(* PLC project Generated.project, CODESYS CODESYS V3.5 SP19 Patch 1 *)
(* stored: creationDateTime 2026-08-18T15:58:35.301546, modificationDateTime 2026-08-18T15:58:35.301546 *)

TYPE ST_ChainBucket : STRUCT
  Idx101_BucketIsOpen : BOOL;  (* 1 = Benne Mécaniquement Ouvert | 0 = Non Confirmé *)
  Idx102_BucketIsClosed : BOOL;  (* 1 = Benne Mécaniquement Fermé | 0 = Non Confirmé *)
  Idx103_OffsetPos_M : REAL;  (* [mètres] Écart d'Ouverture Câble M1/M2 *)
  Idx104_AutoSeqActive : BOOL;  (* : 1 = Séquencement auto (ouverture/fermeture armée par mouvement couplé) en cours *)
  Idx105_StateIncoherent : BOOL;  (* : 1 = État ouvert/fermé INCONNU (ni IsOpen ni IsClosed fiable) -- cause fréquente de blocage *)
  Idx106_FBState : E_State;  (* : État machine FB_Bucket (READY/BUSY/DONE/DISABLED) *)
  Idx107_LastPosM2Open_M : REAL;  (* : Dernière position M2 mémorisée "ouvert" *)
  Idx108_LastPosM2Close_M : REAL;  (* : Dernière position M2 mémorisée "fermé" *)
  Idx109_BucketTooOpen : BOOL;  (* ⚠️ Dépassement ouverture : Delta < OffsetOpen - Tolerance (Enrouler M2) *)
  Idx110_BucketTooClosed : BOOL;  (* ⚠️ Dépassement fermeture : Delta > OffsetClose + Tolerance (Dérouler M2) *)
  Idx111_BucketIsIntermediate : BOOL;  (* ↔️ Position intermédiaire (entrebâillée entre ouvert et fermé) *)
  Idx112_DeltaPosition_M : REAL;  (* 📏 Écart réel signé M2 - M1 (mètres) en direct *)
  Idx201_HmiCmd_BtnOpen : BOOL;  (* 1 = Demande Ouverture IHM | 0 = Relâché *)
  Idx202_HmiCmd_BtnClose : BOOL;  (* 1 = Demande Fermeture IHM | 0 = Relâché *)
  Idx203_CycleCmd_Open : BOOL;  (* 1 = Demande Ouverture par le Cycle Auto *)
  Idx204_CoupledDiveOpenArmed : BOOL;  (* : 1 = Ouverture auto armée (descente couplée demandée, benne pas ouverte) *)
  Idx205_CoupledAscentCloseArmed : BOOL;  (* : 1 = Fermeture auto armée (montée couplée demandée, benne pas fermée) *)
  Idx206_CloseReqActive : BOOL;  (* : 1 = Fermeture mémorisée/en cours (instBucket.CloseReq -- reste à 1 si recul partiel non terminé) *)
  Idx207_OpenReqActive : BOOL;  (* : 1 = Ouverture mémorisée/en cours (instBucket.OpenReq -- idem) *)
  Idx208_MotionBlockedByBucket : BOOL;  (* : 1 = Mouvement couplé BLOQUÉ (auto-séquencement armé mais benne pas Busy -- vérifier Idx306_ErrorIdRaw) *)
  Idx301_EmergencyChainClosed : BOOL;  (* 1 = Boucle Urgence OK | 0 = AU Appuyé *)
  Idx302_BucketFaultActive : BOOL;  (* 0 = Sain | 1 = Défaut Mouvement Benne *)
  Idx303_KoboldAutoStopEnabled : BOOL;  (* 1 = Toggle IHM arrêt auto descente actif *)
  Idx304_KoboldImmersionConfirmed : BOOL;  (* : 1 = Immersion confirmée (front Kobold dans la fenêtre) *)
  Idx305_KoboldBottomTouchLatched : BOOL;  (* : 1 = Fond détecté, descente bloquée (ProcessPermitM1/M2_Descend) *)
  Idx306_ErrorIdRaw : WORD;  (* : bitfield brut FB_Bucket (bit0 timeout, bit1 incohérence, bit2 limites, bit3 codeur non référencé, bit4 glissement M1) *)
  Idx401_BucketBusy : BOOL;  (* 1 = Mouvement Mâchoires en cours | 0 = Repos *)
  Idx402_BucketDone : BOOL;  (* 1 = Position Cible Atteinte | 0 = En cours *)
  Idx403_ControlAscentActive : BOOL;  (* : 1 = Phase vitesse contrôlée montée en cours (post-fermeture auto) *)
  Idx501_M2_CmdRev_DQ : BOOL;  (* 1 = Relais Action Benne M2 ON *)
END_STRUCT;
END_TYPE

TYPE ST_ChainContextGlobal : STRUCT
  Idx101_ModeActive : E_Mode;  (* Mode de marche actif (MANUEL, SEMI_AUTO, MAINT_N1, MAINT_N2) *)
  Idx102_SimulationEnabled : BOOL;  (* 0 = Matériel Réel (Nominal) | 1 = SIMULATION ACTIVE ⚠️ *)
  Idx103_JoystickCommOk : BOOL;  (* 1 = Comm CANopen Joystick OK (Sain) | 0 = Perte Comm CAN *)
  Idx201_JoystickSelected : BOOL;  (* 1 = Pilotage par Joystick Hall | 0 = Pilotage par Boutons IHM *)
  Idx202_BypassNetworkGlobal : BOOL;  (* 0 = Comm Réseau OK | 1 = BYPASS RÉSEAU ACTIF ⚠️ *)
  Idx203_BypassSensorsGlobal : BOOL;  (* 0 = Capteurs Actifs | 1 = AU MOINS 1 CAPTEUR SHUNTÉ ⚠️ *)
  Idx301_EmergencyChainClosed : BOOL;  (* 1 = Boucle AU Matérielle Fermée (OK) | 0 = AU APPUYÉ *)
  Idx302_PowerContactorEngaged : BOOL;  (* 1 = Puissance Armée | 0 = Puissance Coupée *)
  Idx303_SafeStopActiveAny : BOOL;  (* 0 = Sain | 1 = AU MOINS UN SAFESTOP MÉTIER ACTIF *)
  Idx304_PowerCutOffActiveAny : BOOL;  (* 0 = Sain | 1 = COUPURE GENERAL COLLAGE ACTIVEE *)
  Idx401_HmiHeartbeatOk : BOOL;  (* 1 = Liaison IHM Active | 0 = Perte Liaison IHM *)
  Idx402_CycleAutoBusy : BOOL;  (* 1 = Séquenceur Auto en Cours | 0 = Repos *)
END_STRUCT;
END_TYPE

(* ======================================================================= 🔄 ST_ChainCycleSemiAuto — Diagnostic chronologique Séquenceur Semi-Auto ─────────────────────────────────────────────────────────────── 🎯 Rôle : Vue dépannage / Watch CODESYS pour le cycle semi-automatique 📄 Doc métier : DOC/AF/AF_Partie-14_Fonction_Troubleshooting/FB_TroubleshootingView_v1.2.md 🔒 Sécurité : 100% lecture seule / diagnostic d'observation ======================================================================= *)
TYPE ST_ChainCycleSemiAuto : STRUCT
  Idx101_ModeSemiAutoActive : BOOL;  (* 🚦 1. Conditions d'engagement et autorisations 1 = Mode arbitré SEMI_AUTO actif | 0 = Autre mode *)
  Idx102_PowerAndSafetyOk : BOOL;  (* 1 = Chaîne de sécurité OK (PowerContactorEngaged) *)
  Idx103_HeartbeatIhmOk : BOOL;  (* 1 = Liaison IHM<->PLC valide *)
  Idx104_DeadmanArmed : BOOL;  (* 1 = Bouton homme-mort armé (fenêtre 3s active) *)
  Idx105_MancheDeflechi : BOOL;  (* 1 = Permis mouvement armé (manche hors zone neutre) *)
  Idx106_HomedM1M2 : BOOL;  (* 1 = Codeurs treuils M1 et M2 référencés *)
  Idx107_StartCycleRequest : BOOL;  (* 1 = Demande Start reçue (IHM) *)
  Idx108_AbortCycleRequest : BOOL;  (* 1 = Demande Abort reçue (IHM) *)
  Idx201_Ready : BOOL;  (* 🔄 2. État du Séquenceur 1 = Séquenceur prêt à démarrer *)
  Idx202_Busy : BOOL;  (* 1 = Cycle en cours d'exécution *)
  Idx203_Done : BOOL;  (* 1 = Cycle terminé avec succès *)
  Idx204_Error : BOOL;  (* 1 = Défaut ou anomalie bloquante sur le cycle *)
  Idx205_ErrorId : WORD;  (* Code d'erreur interne FB_Cycle *)
  Idx206_Step : E_CycleStep;  (* Étape courante (X0 à X13 + STABILIZING) *)
  Idx207_StepStr : STRING(40);  (* Libellé explicite de l'étape *)
  Idx208_StepAtError : E_CycleStep;  (* Étape mémorisée lors du dernier défaut *)
  Idx301_TargetPosition : INT;  (* 🎯 3. Consignes & Feedbacks Opérationnels Cible translation sélectionnée (1=Trémie, 3=P1) *)
  Idx302_TargetDepth_M : REAL;  (* Profondeur de consigne (m) *)
  Idx303_KoboldBottomTouch : BOOL;  (* 1 = Détection contact fond Kobold *)
  Idx304_SpeedMismatchActive : BOOL;  (* 1 = Alerte écart de vitesse M1/M2 active *)
  Idx305_LimitLegalReached : BOOL;  (* 1 = Limite légale atteinte (descente bloquée) *)
  Idx306_WinchSyncError : BOOL;  (* 1 = Erreur de synchronisme M1/M2 *)
END_STRUCT;
END_TYPE

TYPE ST_ChainDredgingAssist : STRUCT
  Idx101_EnableDiveSearch : BOOL;  (* 1 = Assistance Plongée Armée (IHM) | 0 = Désarmée *)
  Idx102_EnableExtractionSequence : BOOL;  (* 1 = Assistance Extraction Armée (IHM) | 0 = Désarmée *)
  Idx103_EnableDumpAtTremie : BOOL;  (* 1 = Mode Vidage Trémie Armé (IHM) | 0 = Désarmé *)
  Idx201_DiveReady : BOOL;  (* 1 = Assistance Plongée Prête | 0 = Non Prête *)
  Idx202_DiveBusy : BOOL;  (* 1 = Séquence Plongée En Cours | 0 = Repos *)
  Idx203_DiveDone : BOOL;  (* 1 = Fond Confirmé | 0 = En Cours *)
  Idx204_DiveState : E_DiveSearchState;  (* État interne séquenceur plongée *)
  Idx205_DiveError : BOOL;  (* 0 = Sain | 1 = Défaut Plongée *)
  Idx206_DiveErrorId : WORD;  (* bit0: préconditions, bit1: séquence Kobold, bit2: config seuils *)
  Idx207_BottomTouchConfirmed : BOOL;  (* 1 = Contact Fond Confirmé (Kobold ou manuel) | 0 = Non Confirmé *)
  Idx301_ExtractionReady : BOOL;  (* 1 = Assistance Extraction Prête | 0 = Non Prête *)
  Idx302_ExtractionBusy : BOOL;  (* 1 = Séquence Extraction En Cours | 0 = Repos *)
  Idx303_ExtractionDone : BOOL;  (* 1 = Extraction Terminée | 0 = En Cours *)
  Idx304_ExtractionState : E_ExtractionSequenceState;  (* État interne séquenceur extraction *)
  Idx305_ExtractionError : BOOL;  (* 0 = Sain | 1 = Défaut Extraction *)
  Idx306_ExtractionErrorId : WORD;  (* bit0: fond absent, bit1: fermeture, bit2: contrôle remontée, bit3: config *)
  Idx401_OperatorActionId : WORD;  (* Identifiant consigne opérateur conduite (0 = aucune) *)
  Idx402_OperatorAction : STRING(120);  (* Texte consigne opérateur (secours affichage) *)
  Idx501_DumpAtTremieArmed : BOOL;  (* 1 = Bit IHM TglEnableDumpAtTremie actif | 0 = Désarmé *)
  Idx502_DumpAtTremieAssistActive : BOOL;  (* 1 = Mode réellement actif (armé ET Mode MAINT_N1/N2) | 0 = Inactif *)
  Idx503_DumpAtTremieAtTremie : BOOL;  (* 1 = M3 à la position Trémie | 0 = Ailleurs *)
  Idx504_DumpAtTremieBucketOpenArmed : BOOL;  (* 1 = Ouverture benne armée par ce mode | 0 = Non armée *)
  Idx505_DumpAtTremieDescentLocked : BOOL;  (* 1 = Descente M1/M2 verrouillée (M3 hors P1/Maintenance) | 0 = Libre *)
  Idx601_BypassDiveActive : BOOL;  (* 1 = Bypass séquence DiveSearch armé (IHM) *)
  Idx602_BypassKoboldBottomTouched : BOOL;  (* 1 = Fond confirmé par le bypass (front montant Kobold en descente) *)
END_STRUCT;
END_TYPE

TYPE ST_ChainTranslation : STRUCT
  Inputs_100 : ST_Chain_Translation_Inputs;
  Demandes_200 : ST_Chain_Translation_Demandes;
  Safety_300 : ST_Chain_Translation_Safety;
  Control_400 : ST_Chain_Translation_Control;
  Outputs_500 : ST_Chain_Translation_Outputs;
END_STRUCT;
END_TYPE

TYPE ST_ChainWinch : STRUCT
  Inputs_100 : ST_Chain_Winch_Inputs;
  Demandes_200 : ST_Chain_Winch_Demandes;
  Safety_300 : ST_Chain_Winch_Safety;
  Control_400 : ST_Chain_Winch_Control;
  Outputs_500 : ST_Chain_Winch_Outputs;
END_STRUCT;
END_TYPE

TYPE ST_ChainWinchSync : STRUCT
  Idx101_M1_CablePos_M : REAL;  (* [mètres] Position Câble M1 Retenue *)
  Idx102_M2_CablePos_M : REAL;  (* [mètres] Position Câble M2 Benne *)
  Idx103_SyncDelta_M : REAL;  (* [mètres] Écart Relatif M1 - M2 *)
  Idx201_JoyYRaw_Pct : REAL;  (* [%] Consigne Joystick Axe Y (-100% à +100%) *)
  Idx202_SyncEnabled_IHM : BOOL;  (* 1 = Couplage Synchro Actif (Nominal) | 0 = Découplé ⚠️ *)
  Idx203_ArbitratedSpeed_Pct : REAL;  (* [%] Consigne Vitesse Synchro Arbitrée *)
  Idx301_EmergencyChainClosed : BOOL;  (* 1 = Boucle Urgence OK | 0 = Arrêt Urgence *)
  Idx302_SyncFaultActive : BOOL;  (* 0 = Synchro OK | 1 = Écart Synchro Bloquant *)
  Idx303_M1_AscentPermit : BOOL;  (* 1 = Montée M1 Autorisée | 0 = Bloquée (Fdc/Safety) *)
  Idx304_M2_AscentPermit : BOOL;  (* 1 = Montée M2 Autorisée | 0 = Bloquée (Fdc/Safety) *)
  Idx401_SyncMotionAllowed : BOOL;  (* 1 = Mouvement Synchro Autorisé | 0 = Bloqué *)
  Idx402_M1_SetpointSpeed_Pct : REAL;  (* [%] Consigne Vitesse Calculée M1 *)
  Idx403_M2_SetpointSpeed_Pct : REAL;  (* [%] Consigne Vitesse Calculée M2 *)
  Idx501_M1_CmdRelayFwd_DQ : BOOL;  (* 1 = Montée M1 ON | 0 = OFF *)
  Idx502_M2_CmdRelayFwd_DQ : BOOL;  (* 1 = Montée M2 ON | 0 = OFF *)
END_STRUCT;
END_TYPE

(* ═══════════════════════════════════════════════════════════════ 🏗️ ST_HardwareImage — Structure globale d'image matérielle (Frontière HwIn) ─────────────────────────────────────────────────────────────── 🎨 Agrège les 4 sous-domaines matériels : Winch, Translation, Operator, Machine. ═══════════════════════════════════════════════════════════════ *)
TYPE ST_HardwareImage : STRUCT
  Winch : ST_HwWinch;  (* Entrées brutes domaine Treuils M1/M2 + codeurs *)
  Translation : ST_HwTranslation;  (* Entrées brutes domaine Translation M3 + variateur *)
  Operator : ST_HwOperator;  (* Entrées brutes domaine Opérateur / Joystick / bus CAN *)
  Machine : ST_HwMachine;  (* Entrées brutes domaine Sécurités/Communs Machine *)
END_STRUCT;
END_TYPE

(* ═══════════════════════════════════════════════════════════════ 🎯 ST_HomingChecklist — Diagnostic chronologique de référencement (Dépannage) ─────────────────────────────────────────────────────────────── 🎨 Permet de localiser immédiatement l'étape qui bloque le Homing (M1/M2). ═══════════════════════════════════════════════════════════════ *)
TYPE ST_HomingChecklist : STRUCT
  Step1_ModeAuthorized : BOOL;  (* 1. Pré-requis de mode TRUE = Mode MAINT_N1 ou MAINT_N2 actif ➔ Commutateur Mode IHM : GVL_IHM.Modes *)
  Step2_WinchSelected : BOOL;  (* TRUE = Treuil sélectionné en MAINT_N2 ➔ Bouton IHM : GVL_IHM.Modes.Cmd.TglJoystickMaster / Selection Treuil *)
  Step3_EncoderAvailable : BOOL;  (* 2. Santé Matériel & Bus TRUE = Codeur EtherCAT OK & E/S OK ➔ Si simu : GVL_Simulation.SimWinchActive=1 / SimSafetyActive=1 *)
  HwIn_ContactorsReleased_DI : BOOL;  (* 2bis. Entrées physiques directes HwIn (vérité terrain) Retours contacteurs retombés issus de HwIn.Winch *)
  HwIn_BrakeIsOpen_DI : BOOL;  (* Retour fin de course frein (1 = ouvert) issu de HwIn.Winch *)
  HwIn_TopPositionFree_DI : BOOL;  (* Capteur position haute commun libre (1 = libre) issu de HwIn.Winch *)
  Step4_ContactorsReleased : BOOL;  (* 3. État Physique Machine TRUE = Tous les contacteurs retombés (attendre l'arrêt complet) *)
  Step5_BrakeApplied : BOOL;  (* TRUE = Frein serré (attendre l'arrêt complet) *)
  TopPositionSensorActive : BOOL;  (* 📍 Fin de course haut physique (TRUE = au contact) *)
  BucketIsOpen : BOOL;  (* 🪣 Benne Ouvert (TRUE = Ouvert) ➔ Pour forcer sans codeur : GVL_IHM.M2TreuilBenne.Bucket.Cmd.BtnConfirmOpenPos *)
  AllConditionsMet : BOOL;  (* 4. Séquence & Bilan TRUE = Prêt pour le homing ! ➔ Déclencher : GVL_IHM.M1TreuilRetenue.Cmd.BtnHome (à 8m) ou BtnHomingAtZero (à 0m) *)
  HomingBusy : BOOL;  (* TRUE = Séquence de calage en cours *)
  HomingDone : BOOL;  (* TRUE = Calage réussi *)
  HomingHomed : BOOL;  (* TRUE = Treuil actuellement référencé *)
  HomingSuspect : BOOL;  (* TRUE = Doute redémarrage ➔ Lever le doute via : GVL_IHM.M1TreuilRetenue.Cmd.BtnConfirmCoherence *)
  RejectErrorMask : WORD;  (* 5. Code de rejet exact Bitmask d'erreur FB_Encoder_Homing.ErrorId *)
END_STRUCT;
END_TYPE

(* ═══════════════════════════════════════════════════════════════ 🕹️ ST_JoystickChecklist — Diagnostic chronologique communication & prise en main Joystick ─────────────────────────────────────────────────────────────── 🎨 Permet de vérifier la chaîne Joystick (CANopen, Homme-mort, Neutre, Calibration). ═══════════════════════════════════════════════════════════════ *)
TYPE ST_JoystickChecklist : STRUCT
  Step1_CanBusActive : BOOL;  (* 1. Bus & Matériel TRUE = Bus CANopen en état ACTIVE *)
  Step2_JoystickOperational : BOOL;  (* TRUE = Esclave JOY1 en état RUNNING *)
  HwIn_JoyBtnRaw_DI : BOOL;  (* 1bis. Entrées physiques directes HwIn Bouton brut homme-mort issu de HwIn.Operator *)
  NeutralXAct : BOOL;  (* TRUE = Axe X au neutre (PRG_02_Acquisition.JoystickXNeutral) *)
  NeutralYAct : BOOL;  (* TRUE = Axe Y au neutre (PRG_02_Acquisition.JoystickYNeutral) *)
  Step3_DeadmanPressed : BOOL;  (* 2. Prise en main & Sécurité TRUE = Bouton Homme-Mort appuyé *)
  Step4_NeutralAcquired : BOOL;  (* TRUE = Repassé par le neutre (autorisation mouvement) *)
  DeadmanArmed : BOOL;  (* TRUE = Homme-Mort armé avec passage au neutre validé *)
  AllConditionsMet : BOOL;  (* 3. Éligibilité globale TRUE = Joystick prêt pour piloter un axe *)
  JoystickSelected : BOOL;  (* TRUE = Joystick maître sélectionné IHM *)
  SelJoystickWinch : INT;  (* Sélection Treuil (0=Couplé M1+M2, 1=M1 seul, 2=M2 seul) *)
  RawX : INT;  (* 4. Mesures brutes & Filtrées Valeur brute axe X (0..10000) *)
  RawY : INT;  (* Valeur brute axe Y (0..10000) *)
  DeflectionX_Pct : REAL;  (* Déflexion signée X (%) *)
  DeflectionY_Pct : REAL;  (* Déflexion signée Y (%) *)
  DirectionX : INT;  (* Direction filtrée X (-1 / 0 / +1) *)
  DirectionY : INT;  (* Direction filtrée Y (-1 / 0 / +1) *)
END_STRUCT;
END_TYPE

(* ═══════════════════════════════════════════════════════════════ ⚙️ ST_MotionChecklist — Diagnostic chronologique de commande de mouvement ─────────────────────────────────────────────────────────────── 🎨 Permet de voir en un coup d'œil pourquoi un ordre de mouvement ne fait pas coller les relais. ═══════════════════════════════════════════════════════════════ *)
TYPE ST_MotionChecklist : STRUCT
  Step1_PowerEngaged : BOOL;  (* 1. Puissance & Mode TRUE = Contacteur principal sous tension (PowerContactorEngaged_DI) ➔ Armer puissance via Reset *)
  Step2_ModeAuthorized : BOOL;  (* TRUE = Mode MAINT_N1 ou N2 actif (pas DISABLE) ➔ Commutateur Mode IHM *)
  Step3_NotBusyOtherTask : BOOL;  (* TRUE = Pas d'autre séquence en cours (Homing, Benne busy, etc.) *)
  HwIn_PowerContactorEngaged_DI : BOOL;  (* 1bis. Entrées physiques directes HwIn (vérité terrain) Contacteur puissance principal issu de HwIn.Machine *)
  HwIn_BrakeIsOpen_DI : BOOL;  (* Retour fin de course frein (1 = ouvert) issu de HwIn *)
  Cmd_BrakeRelease : BOOL;  (* Ordre de commande d'ouverture de frein généré par l'automate *)
  Step4_MotionRequested : BOOL;  (* 2. Intention & Demande TRUE = Demande active (Bouton IHM ou Joystick) ➔ Si IHM : TglJoystickMaster doit être à 0 ! *)
  RequestedDirection : INT;  (* +1 = Montée, -1 = Descente, 0 = Repos *)
  RequestedSpeedPct : REAL;  (* 0..100 % consigne demandée *)
  Step5_NoSafetyFault : BOOL;  (* 3. Chaîne de Sécurité & Verrous TRUE = Pas de SafeStop ni AU actif sur cet axe *)
  Step6_DirectionAllowed : BOOL;  (* TRUE = Sens autorisé (AscentPermit/DescendPermit) *)
  Step7_BrakeReleased : BOOL;  (* TRUE = Commande frein activée & retour frein OK *)
  Step8_OutputInterlockOk : BOOL;  (* TRUE = Étage de sortie LD débloqué (pas d'interlock actif) *)
  AllConditionsMet : BOOL;  (* 4. Bilan & Exécution Physiques 🟢 TRUE = TOUTES LES CONDITIONS SONT REMPLIES, LES RELAIS DOIVENT COLLER ! *)
  RelayFwdActive : BOOL;  (* 🛗 Relais Montée physiquement commandé *)
  RelayRevActive : BOOL;  (* 🛗 Relais Descente physiquement commandé *)
  SpeedContactor1Active : BOOL;  (* 🔌 Contacteur de vitesse Palier 1 commandé *)
END_STRUCT;
END_TYPE

(* ═══════════════════════════════════════════════════════════════ 🛡️ ST_SafetyChecklist — Diagnostic chronologique réarmement chaîne de sécurité / AU ─────────────────────────────────────────────────────────────── 🎨 Permet d'identifier immédiatement pourquoi la puissance / AU ne réarme pas. ═══════════════════════════════════════════════════════════════ *)
TYPE ST_SafetyChecklist : STRUCT
  SimulationModeActive : BOOL;  (* 0. Aiguillage source — dit QUELLE entree alimente les steps 1-3 ci-dessous. Absent jusqu'ici : diagnostiquer un blocage AU en full simu obligeait a rouvrir GVL_Simulation dans un Watch separe (, banc sans HW). TRUE = bit maitre simu actif (GVL_Simulation.SimulationModeActive) *)
  SimSafetyActive : BOOL;  (* TRUE = domaine Safety simule ➔ Step1-3 lisent FB_Sim_Safety, pas les DI/comm reelles *)
  HwIn_EmergencyChainClosed_DI : BOOL;  (* 0bis. Entrées physiques directes HwIn (vérité terrain) Boucle AU physique ou simulée issue de HwIn.Machine *)
  HwIn_PowerContactorEngaged_DI : BOOL;  (* Retour contacteur de puissance issu de HwIn.Machine *)
  HwIn_EmergencyBtnCut_HMI : BOOL;  (* Commande coupure AU IHM *)
  Step1_InputModulesOk : BOOL;  (* 1. Intégrité matérielle & modules E/S TRUE = Les 3 cartes E/S physiques sont RUNNING ➔ En simu : GVL_Simulation.SimSafetyActive=1 *)
  Step2_EmergencyBtnNotCut : BOOL;  (* TRUE = Pas d'appui AU ➔ Déverrouiller le BP coup-de-poing physique ou IHM : GVL_IHM.Modes.Cmd.BtnEmergencyCutOff *)
  Step3_EmergencyChainClosed : BOOL;  (* TRUE = Boucle physique AU fermée (EmergencyChainClosed_DI) *)
  Step4_ContactorReleased : BOOL;  (* 2. Conditions de réarmement TRUE = Contacteur relâché ; précondition AF01 avant réarmement *)
  Step5_ArmingAllowed : BOOL;  (* TRUE = Armable ; acquitter si nécessaire puis générer un front BtnEmergencyArming *)
  ArmingStep : INT;  (* 3. Séquence de réarmement 0=IDLE, 1=TestA, 2=RestoreA, 3=TestB, 4=RestoreB, 5=Pulse, 6=Confirm *)
  ArmingPulseActive : BOOL;  (* TRUE = Impulsion d'armement en cours *)
  ArmingBusy : BOOL;  (* TRUE = séquence de réarmement ou verrouillage en cours *)
  LockoutActive : BOOL;  (* TRUE = verrouillage temporel entre tentatives *)
  PowerContactorEngaged : BOOL;  (* TRUE = Contacteur principal sous tension (PowerContactorEngaged_DI) *)
  PowerCutOffActive : BOOL;  (* TRUE = demande de coupure safety active *)
  PowerCutOffRequest : BOOL;  (* TRUE = demande de coupure AU (entrée instSafetyEmergencyManagement) *)
  MaintainAActive : BOOL;  (* TRUE = maintien voie A demandé *)
  MaintainBActive : BOOL;  (* TRUE = maintien voie B demandé *)
  AllConditionsMet : BOOL;  (* TRUE = état final : chaîne OK et puissance engagée *)
  SafetyError : BOOL;  (* 4. Erreurs TRUE = Défaut sécurité actif *)
  ArmingErrorId : WORD;  (* bit0 redondance ; bit1 échec confirmation contacteur *)
  RedundancyTestFailed : BOOL;  (* TRUE = Défaut test de redondance contacteurs *)
  ArmingFailed : BOOL;  (* TRUE = Échec de la séquence d'armement *)
END_STRUCT;
END_TYPE

(* values of E_State: DISABLED: Enable faux, neutralisé; INIT: Démarrage / vérifs; READY: Prêt, attend ordre; BUSY: Action en cours; DONE: Action terminée; STOPPING: Décél rampe avant arrêt (StartStop=FALSE ou SafeStop=TRUE) *)

{attribute 'qualified_only'}
{attribute 'strict'}
TYPE E_State : (DISABLED := 0, INIT := 1, READY := 2, BUSY := 3, DONE := 4, STOPPING := 5);
END_TYPE

(* values of E_Mode: DISABLE: Mode Désactivé / Veille de sécurité (sorties bloquées); MAINT_N1: Manuel Niveau 1 : Pilotage unitaire avec toutes sécurités actives; MAINT_N2: Manuel Niveau 2 : Pilotage dégradé (droits étendus + bypasses autorisés); SEMI_AUTO: Mode Semi-Automatique (séquenceur automatique) *)

{attribute 'qualified_only'}
{attribute 'strict'}
TYPE E_Mode : (DISABLE := 0, MAINT_N1 := 1, MAINT_N2 := 2, SEMI_AUTO := 3);
END_TYPE

(* values of E_CycleStep: X0_PREPARATION: Début de graphe : à la TRÉMIE, treuils en position HAUTE; X1_HOMING: Vitesses lentes pour chercher capteur top + référencement; X2_WORK_POS_SELECT: Sélection cible Trémie/P1/Maintenance + translation validée; X3_OPEN_BUCKET: Ouverture benne (si déjà ouverte -> passe vite); X4_DESCEND_OPEN: Plongée benne ouverte, M1+M2 synchro, Kobold mesure ON; X5_BOTTOM_CONFIRMED: Fond validé (FB_DiveSearch) ; arrêt descente; X6_CLOSE_BUCKET: Fermeture benne — tolérance « à peu près fermé »; X7_CTRL_ASCENT: Remontée palier 1 de contrôle; X8_ASCENT_LOADED: Remontée nominale jusqu'à limite haute; X9_DRAIN_PAUSE: Égouttage temporisé — temps affiché IHM; X10_TRANSLATE_DUMP: Translation vers trémie + avertissements IHM; X11_OPEN_DUMP: Ouverture benne = vidage ; montée possible, descente ouvre; X13_DONE_SYNC: Fin de cycle, synchronisation finale (R4) + compteur; STABILIZING: État d'attente/stabilisation — pas une erreur *)

{attribute 'qualified_only'}
{attribute 'strict'}
TYPE E_CycleStep : (X0_PREPARATION := 0, X1_HOMING := 1, X2_WORK_POS_SELECT := 2, X3_OPEN_BUCKET := 3, X4_DESCEND_OPEN := 4, X5_BOTTOM_CONFIRMED := 5, X6_CLOSE_BUCKET := 6, X7_CTRL_ASCENT := 7, X8_ASCENT_LOADED := 8, X9_DRAIN_PAUSE := 9, X10_TRANSLATE_DUMP := 10, X11_OPEN_DUMP := 11, X13_DONE_SYNC := 13, STABILIZING := 14);
END_TYPE

(* values of E_DiveSearchState: WAIT_PRECONDITIONS: Attente benne ouverte, positions et Kobold au repos; READY_TO_DESCEND: Prêt à assister une demande de descente; SEARCHING_IMMERSION: Descente : attente front 0->1 dans fenêtre eau; SEARCHING_BOTTOM: Immersion validée : attente front 1->0 au fond; BOTTOM_CONFIRMED: Fond validé ; extraction peut être demandée; ERROR_HOLD: Séquence invalide, descente assistée interdite *)

{attribute 'qualified_only'}
{attribute 'strict'}
TYPE E_DiveSearchState : (WAIT_PRECONDITIONS := 0, READY_TO_DESCEND := 1, SEARCHING_IMMERSION := 2, SEARCHING_BOTTOM := 3, BOTTOM_CONFIRMED := 4, ERROR_HOLD := 5);
END_TYPE

(* values of E_ExtractionSequenceState: WAIT_BOTTOM_CONFIRMATION: Attente fond Kobold ou attestation opérateur; READY_TO_CLOSE: Prêt à fermer la benne; CLOSING_BUCKET: FB_Bucket ferme M2 seul; CONTROL_ASCENT: M1/M2 synchronisés au palier sans contacteur vitesse; NOMINAL_ASCENT: Montée couplée avec vitesse demandée opérateur; ERROR_HOLD: Défaut extraction, reprise interdite avant reset *)

{attribute 'qualified_only'}
{attribute 'strict'}
TYPE E_ExtractionSequenceState : (WAIT_BOTTOM_CONFIRMATION := 0, READY_TO_CLOSE := 1, CLOSING_BUCKET := 2, CONTROL_ASCENT := 3, NOMINAL_ASCENT := 4, ERROR_HOLD := 5);
END_TYPE

TYPE ST_Chain_Translation_Control : STRUCT
  Idx401_MotionAllowed : BOOL;  (* 1 = Mouvement Translation Autorisé | 0 = Bloqué *)
  Idx402_SetpointFreq_Hz : REAL;  (* [Hz] Consigne Fréquence Calculée *)
  Idx403_DriveControlWord : WORD;  (* Mot de Commande Calculé Variateur AC600 *)
  Idx404_FinalInterlockState : E_State;  (* 🛡️ État frontière _LD *)
  Idx405_FinalInterlockReason : E_TranslationFinalInterlockReason;  (* 🛡️ Cause mémorisée *)
  Idx406_BrakeCommandOpenConfirmed : BOOL;  (* 🔌 Contacteur/bobine, pas frein mécanique *)
  Idx407_BrakeTimeoutElapsed : TIME;  (* ⏱️ Watchdog 500ms écoulé *)
END_STRUCT;
END_TYPE

TYPE ST_Chain_Translation_Demandes : STRUCT
  Idx201_JoyXRaw_ANA : INT;  (* [pts] Bruts Joystick Axe X *)
  Idx202_JoyXScaled_Pct : REAL;  (* [%] Consigne Joystick Axe X (-100% à +100%) *)
  Idx203_HmiCmd_BtnFwd : BOOL;  (* 1 = Bouton Avance IHM | 0 = Relâché *)
  Idx204_HmiCmd_BtnRev : BOOL;  (* 1 = Bouton Recul IHM | 0 = Relâché *)
  Idx205_HmiTargetPosition : INT;  (* Cible Sélectionnée IHM (1=Trémie, 2=P2, 3=P1) *)
  Idx206_CycleTargetPosition : INT;  (* Cible Sélectionnée par le Cycle Auto *)
  Idx207_ModeActive : E_Mode;  (* Mode courant (MANU_N1, AUTO_N1...) *)
  Idx208_BypassNetworkActive : BOOL;  (* 0 = Comm Variateur OK | 1 = Bypass Réseau Actif ⚠️ *)
  Idx209_ArbitratedSpeed_Pct : REAL;  (* [%] Consigne finale Vitesse Translation *)
END_STRUCT;
END_TYPE

TYPE ST_Chain_Translation_Inputs : STRUCT
  Idx101_PosTremie_DI : BOOL;  (* 1 = Position Trémie Atteinte | 0 = Absent *)
  Idx102_PosPV_DI : BOOL;  (* 1 = Zone Ralentissement PV Atteinte | 0 = Absent *)
  Idx103_PosP2_DI : BOOL;  (* 1 = Position Fosse P2 Atteinte | 0 = Absent *)
  Idx104_PosP1_DI : BOOL;  (* 1 = Position Fosse P1 Atteinte | 0 = Absent *)
  Idx105_PosMaintenance_DI : BOOL;  (* 1 = Position Service Maintenance Atteinte | 0 = Absent *)
  Idx106_DriveActualFreq_Hz : REAL;  (* [Hz] Fréquence Réelle Mesurée Variateur *)
  Idx107_DriveStatusWord : WORD;  (* Mot d'état Brut Variateur AC600 *)
  Idx108_BrakeApplied : BOOL;  (* TRUE = frein SERRÉ (NOT BrakeFeedback — IHM garde le sens serré) *)
  Idx109_DriveThermalOk : BOOL;  (* TRUE = thermique moteur/variateur AC600 OK (diagnostic seul) *)
END_STRUCT;
END_TYPE

TYPE ST_Chain_Translation_Outputs : STRUCT
  Idx501_CmdDriveControlWord : WORD;  (* Mot de Commande Transmis EtherCAT AC600 *)
  Idx502_CmdDriveFreq_Hz : UINT;  (* [0.01Hz] Consigne Fréquence Transmise EtherCAT *)
  Idx503_CmdBrakeRelease_RQ : BOOL;  (* 1 = Bobine Frein Translation Alimentée (Ouvert) *)
END_STRUCT;
END_TYPE

TYPE ST_Chain_Translation_Safety : STRUCT
  Idx301_EmergencyChainClosed : BOOL;  (* 1 = Boucle Urgence OK | 0 = Arrêt d'Urgence Appuyé *)
  Idx302_SafeStopActive : BOOL;  (* 0 = Sain (Autorisé) | 1 = Arrêt Rapide Translation *)
  Idx303_PowerCutOffActive : BOOL;  (* 0 = Puissance OK | 1 = Coupure Puissance *)
  Idx304_LimitSwitchFwdActive : BOOL;  (* 0 = Sain | 1 = Fin de Course Extrême Avance *)
  Idx305_LimitSwitchRevActive : BOOL;  (* 0 = Sain | 1 = Fin de Course Extrême Recul *)
  Idx306_BypassLimitSwitch : BOOL;  (* 0 = Fins de course actives | 1 = Shuntés IHM ⚠️ *)
  Idx307_PositionDecoderIncoherent : BOOL;  (* 0 = Décodage 5 Capteurs OK | 1 = Incohérence Position *)
  Idx308_HeightInterlockBlocking : BOOL;  (* : 0 = M1 ET M2 ≥ hauteur mini (ou bypass) | 1 = Translation bloquée (risque collision) *)
  Idx309_ErrorOperatorComm : BOOL;  (* Défauts safety déchiffrés (bits ErrorId) — visibles individuellement à l'IHM bit0 Perte communication opérateur (joystick CAN / heartbeat IHM) *)
  Idx310_ErrorDriveComm : BOOL;  (* bit1 Perte communication EtherCAT variateur *)
  Idx311_ErrorPhaseRotation : BOOL;  (* bit2 Mauvaise rotation de phases *)
  Idx312_ErrorBrakeThermal : BOOL;  (* bit3 Surchauffe thermique frein commun *)
  Idx313_ErrorMecaB : BOOL;  (* bit4 Absence confirmation arrêt *)
  Idx314_ErrorMecaA : BOOL;  (* bit5 Mouvement non commandé *)
  Idx315_ErrorLimitSwitch : BOOL;  (* bit6 Limite extrême atteinte *)
  Idx316_ErrorSensorIncoherent : BOOL;  (* bit7 Mot capteurs position incohérent *)
END_STRUCT;
END_TYPE

TYPE ST_Chain_Winch_Control : STRUCT
  Idx401_MotionAllowed : BOOL;  (* 1 = Prêt / Mouvement Autorisé | 0 = Bloqué *)
  Idx402_SpeedStepCalculated : INT;  (* Palier Vitesse Calculé (0, 1, 2, 3, 4) *)
  Idx403_SpeedRamp_Pct : REAL;  (* [%] Consigne Vitesse après Rampe *)
  Idx404_BrakeReleaseAuthorized : BOOL;  (* 1 = Ordre Ouverture Frein | 0 = Ordre Serrage *)
  Idx405_FinalInterlockState : E_WinchFinalInterlockState;  (* 🛡️ État frontière _LD *)
  Idx406_FinalInterlockReason : E_WinchFinalInterlockReason;  (* 🛡️ Cause mémorisée *)
  Idx407_FinalAuthorizedStep : INT;  (* 🪜 Palier réellement autorisé *)
  Idx408_BrakeCommandOpenConfirmed : BOOL;  (* 🔌 Contacteur/bobine, pas frein mécanique *)
  Idx409_BrakeTimeoutElapsed : TIME;  (* ⏱️ Watchdog 500ms écoulé *)
  Idx410_RestartDelayElapsed : TIME;  (* ⏱️ Verrou 900ms écoulé *)
  Idx411_StepDelayElapsed : TIME;  (* ⏱️ Délai palier 1s250 écoulé *)
  Idx412_InTopSlowdownZone : BOOL;  (* : Palier plafonné à 1, approche limite haute *)
  Idx413_InBottomSlowdownZone : BOOL;  (* : Palier plafonné à 1, approche limite basse (câble ou légale) *)
  Idx414_BottomLimitActiveM : REAL;  (* : Limite basse active (m) — câble physique OU légale, la plus restrictive *)
END_STRUCT;
END_TYPE

TYPE ST_Chain_Winch_Demandes : STRUCT
  Idx201_JoyRawPhysical_ANA : INT;  (* [pts] Bruts convertisseur (-2048 à +2048) *)
  Idx202_JoyScaledPhysical_Pct : REAL;  (* [%] Consigne Joystick (-100% à +100%) *)
  Idx203_HmiManualCmd_BtnUp : BOOL;  (* 1 = Appui Bouton Montée IHM | 0 = Relâché *)
  Idx204_HmiManualCmd_BtnDown : BOOL;  (* 1 = Appui Bouton Descente IHM | 0 = Relâché *)
  Idx205_CycleAutoCmd_Pct : REAL;  (* [%] Consigne auto envoyée par le Cycle *)
  Idx206_ModeActive : E_Mode;  (* Mode courant (MANU_N1, AUTO_N1, MAINT_N2...) *)
  Idx207_BypassOperatorComm : BOOL;  (* 0 = Comm Normale OK | 1 = Bypass Réseau Actif ⚠️ *)
  Idx208_ArbitratedSpeed_Pct : REAL;  (* [%] Consigne finale retenue après arbitrage *)
  Idx209_ArbitratedDirection : INT;  (* +1 = Montée | 0 = Neutre | -1 = Descente *)
  Idx210_CoupledUserRequestDirection : INT;  (* +1 = Montée | 0 = Neutre | -1 = Descente *)
  Idx211_CoupledUserRequestActive : BOOL;  (* 1 = demande utilisateur couplée active *)
END_STRUCT;
END_TYPE

TYPE ST_Chain_Winch_Inputs : STRUCT
  Idx101_EncoderRawPos : DINT;  (* [Valeur brutes pts] Codeur connecté *)
  Idx102_CablePos_M : REAL;  (* [mètres] Position calculée du câble *)
  Idx103_ContactorsReleased_DI : BOOL;  (* 1 = OK (Tous contacteurs retombés à l'arrêt) | 0 = Contacteur collé *)
  Idx104_BrakeApplied : BOOL;  (* TRUE = frein SERRÉ (NOT BrakeFeedback — IHM garde le sens serré) *)
  Idx105_ThermalOk_DI : BOOL;  (* 1 = Température OK (Sain) | 0 = Surchauffe Moteur M1 *)
END_STRUCT;
END_TYPE

TYPE ST_Chain_Winch_Outputs : STRUCT
  Idx501_CmdRelayFwd_Up_DQ : BOOL;  (* 1 = Relais Montée ON | 0 = OFF *)
  Idx502_CmdRelayRev_Down_DQ : BOOL;  (* 1 = Relais Descente ON | 0 = OFF *)
  Idx503_CmdSpeedContactor1_DQ : BOOL;  (* 1 = Contacteur Vitesse 1 ON | 0 = OFF *)
  Idx504_CmdSpeedContactor4_DQ : BOOL;  (* 1 = Contacteur Vitesse 4 ON (Plein Gaz) | 0 = OFF *)
  Idx505_CmdBrakeRelease_RQ : BOOL;  (* 1 = Bobine Frein Alimentée (Ouvert) | 0 = Non Alimentée (Serré) *)
END_STRUCT;
END_TYPE

TYPE ST_Chain_Winch_Safety : STRUCT
  Idx301_EmergencyChainClosed : BOOL;  (* 1 = Boucle Urgence OK (Armé) | 0 = Arrêt d'Urgence Appuyé *)
  Idx302_SafeStopActive : BOOL;  (* 0 = Sain (Autorisé) | 1 = Arrêt Rapide Métier Actif *)
  Idx303_PowerCutOffActive : BOOL;  (* 0 = Puissance OK | 1 = Coupure Puissance Sécurité *)
  Idx304_TopSensorPhysical_DI : BOOL;  (* 1 = Capteur Haut Libre (Sain) | 0 = Butée Haute Atteinte *)
  Idx305_TopSensorBypassActive : BOOL;  (* 0 = Capteur Actif | 1 = Capteur Haut Shunté IHM ⚠️ *)
  Idx306_AscentPermitEffective : BOOL;  (* 1 = Montée Autorisée | 0 = MONTÉE BLOQUÉE *)
  Idx307_SlackCablePhysical_DI : BOOL;  (* 1 = Câble Tendu (Sain) | 0 = Mou de Câble Détecté *)
  Idx308_SlackCableBypassActive : BOOL;  (* 0 = Capteur Actif | 1 = Mou de Câble Shunté IHM ⚠️ *)
  Idx309_DescendPermitEffective : BOOL;  (* 1 = Descente Autorisée | 0 = DESCENTE BLOQUÉE *)
  Idx310_ErrorOperatorComm : BOOL;  (* Défauts safety déchiffrés (bits ErrorId) — visibles individuellement à l'IHM bit0 Perte communication opérateur (joystick CAN / heartbeat IHM) *)
  Idx311_ErrorEncoder : BOOL;  (* bit1 Perte codeur de ce treuil *)
  Idx312_ErrorPhaseRotation : BOOL;  (* bit4 Mauvaise rotation de phases *)
  Idx313_ErrorMecaA : BOOL;  (* bit7 Mouvement non commandé / roue libre *)
  Idx314_ErrorMecaB : BOOL;  (* bit8 Absence confirmation arrêt sans commande *)
  Idx315_ErrorMecaC : BOOL;  (* bit9 Glissement M1 pendant cycle benne *)
  Idx316_ErrorMecaD : BOOL;  (* bit11 Non-arrêt sur capteur haut *)
  Idx317_ErrorMecaE : BOOL;  (* bit12/13 Écart synchro critique M1/M2 *)
  Idx318_ErrorBrakeThermal : BOOL;  (* bit10 Surchauffe thermique frein commun *)
  Idx319_ErrorOppositeDir : BOOL;  (* bit14 Sens réel opposé au sens commandé *)
  Idx320_ErrorNoMovement : BOOL;  (* bit15 Absence de mouvement malgré commande *)
END_STRUCT;
END_TYPE

(* ═══════════════════════════════════════════════════════════════ 🏗️ ST_HwMachine — Image matérielle brute des entrées communes Machine ─────────────────────────────────────────────────────────────── 🎨 Regroupe les signaux physiques d'entrée bruts communs à la machine. ═══════════════════════════════════════════════════════════════ *)
TYPE ST_HwMachine : STRUCT
  PowerContactorEngaged_DI : BOOL;  (* Confirm. contacteur puissance engagé *)
  EmergencyChainClosed_DI : BOOL;  (* Boucle AU fermée (coup-de-poing + contact PLC) *)
  PhaseRotationOk_DI : BOOL;  (* Contrôle rotation phases élec. OK *)
  M1_M2_M3_BrakeThermalOk_DI : BOOL;  (* Thermique frein M1/M2/M3 commun OK *)
  M1_M2_KoboldBottomTouch_DI : BOOL;  (* Retour détecteur fond Kobold *)
  HydraulicThermalOk_DI : BOOL;  (* Thermique centrale hydraulique OK *)
  ConveyorInfeedReady_DI : BOOL;  (* Autorisation démarrage crible (dépôt gravats) *)
  HopperFull_OR_GateRaised_DI : BOOL;  (* : Trémie pleine OU grille levée — pas encore câblé électriquement, *)
END_STRUCT;
END_TYPE

(* ═══════════════════════════════════════════════════════════════ 🏗️ ST_HwOperator — Image matérielle brute des entrées Opérateur / Joystick ─────────────────────────────────────────────────────────────── 🎨 Regroupe les signaux physiques d'entrée bruts du joystick CANopen JOY1. ═══════════════════════════════════════════════════════════════ *)
TYPE ST_HwOperator : STRUCT
  JoyXRaw_ANA1 : INT;  (* Valeur brute analogique axe X (Translation) *)
  JoyYRaw_ANA2 : INT;  (* Valeur brute analogique axe Y (Levage) *)
  JoyBtnRaw : BOOL;  (* Bouton brut joystick (Homme-Mort) *)
  CanBusState : INT;  (* État bus CANopen (CANbus.GetBusState) *)
  JOY1_DeviceState : DEVICE_STATE;  (* État device JOY1 (GetDeviceState) *)
END_STRUCT;
END_TYPE

(* ═══════════════════════════════════════════════════════════════ 🏗️ ST_HwTranslation — Image matérielle brute des entrées Translation M3 ─────────────────────────────────────────────────────────────── 🎨 Regroupe les signaux physiques d'entrée bruts de la translation M3 (AC600). ═══════════════════════════════════════════════════════════════ *)
TYPE ST_HwTranslation : STRUCT
  M3_PosTremie_DI : BOOL;  (* Capteur position trémie *)
  M3_PosPV_DI : BOOL;  (* Capteur position point de vitesse (pré-ralentissement) *)
  M3_PosPVP2_DI : BOOL;  (* Capteur position P2 / petite vitesse avant P1 *)
  M3_PosP1_DI : BOOL;  (* Capteur position P1 *)
  M3_PosMaintenance_DI : BOOL;  (* Capteur position maintenance *)
  M3_BrakeIsOpen_DI : BOOL;  (* Retour frein M3 (1 = ouvert) *)
  M3_ThermalOK_DI : BOOL;  (* Retour disjoncteur thermique moteur/variateur AC600 (1 = OK) — diagnostic seul, l'AC600 se protège lui-même *)
  M3_StatusWord : WORD;  (* Status word variateur AC600 *)
  M3_ActualFrequencyHz : UINT;  (* Fréquence réelle variateur AC600 (x100) *)
  AC600_DeviceState : DEVICE_STATE;  (* État device AC600 (GetDeviceState) *)
END_STRUCT;
END_TYPE

(* ═══════════════════════════════════════════════════════════════ 🏗️ ST_HwWinch — Image matérielle brute des entrées Treuils M1 / M2 ─────────────────────────────────────────────────────────────── 🎨 Regroupe les signaux physiques d'entrée bruts des treuils M1 et M2. ═══════════════════════════════════════════════════════════════ *)
TYPE ST_HwWinch : STRUCT
  M1_ContactorsReleased_DI : BOOL;  (* Retours contacteurs M1 retombés *)
  M1_ThermalOk_DI : BOOL;  (* Thermique moteur M1 OK *)
  M1_BrakeIsOpen_DI : BOOL;  (* Retour frein M1 (1 = ouvert) *)
  M2_ContactorsReleased_DI : BOOL;  (* Retours contacteurs M2 retombés *)
  M2_ThermalOk_DI : BOOL;  (* Thermique moteur M2 OK *)
  M2_BrakeIsOpen_DI : BOOL;  (* Retour frein M2 (1 = ouvert) *)
  M1M2_TopPositionFree_DI : BOOL;  (* Capteur position haute commun M1/M2 libre *)
  M2_TensionedCable_DI : BOOL;  (* Capteur mou de câble M2 (câble tendu) *)
  COD1_PosValue : UDINT;  (* Valeur brute position codeur COD1 (M1) *)
  COD1_Alarms : UINT;  (* Alarmes brutes COD1 *)
  COD1_Warnings : UINT;  (* Avertissements bruts COD1 *)
  COD1_DeviceState : DEVICE_STATE;  (* État device COD1 (GetDeviceState) *)
  COD2_PosValue : UDINT;  (* Valeur brute position codeur COD2 (M2) *)
  COD2_Alarms : UINT;  (* Alarmes brutes COD2 *)
  COD2_Warnings : UINT;  (* Avertissements bruts COD2 *)
  COD2_DeviceState : DEVICE_STATE;  (* État device COD2 (GetDeviceState) *)
END_STRUCT;
END_TYPE

{attribute 'qualified_only'}
{attribute 'strict'}
TYPE E_TranslationFinalInterlockReason : (NONE := 0, BRAKE_COMMAND_NOT_CONFIRMED := 1, RESTART_INHIBITED := 2);
END_TYPE

(* values of E_WinchFinalInterlockReason: NONE: Aucun blocage actif; BRAKE_COMMAND_NOT_CONFIRMED: Absence confirmation ouverture frein > 500ms; RESTART_INHIBITED: Inhibition redemarrage actif *)

{attribute 'qualified_only'}
{attribute 'strict'}
TYPE E_WinchFinalInterlockReason : (NONE := 0, BRAKE_COMMAND_NOT_CONFIRMED := 1, RESTART_INHIBITED := 2);
END_TYPE

(* values of E_WinchFinalInterlockState: DISABLED: Desactive / Hors service; READY: Pret / Etat nominal; WAIT_BRAKE_COMMAND_CONFIRMATION: Attente confirmation feedback frein; WAIT_STEP_DELAY: Temporisation changement de palier; WAIT_RESTART_DELAY: Temporisation anti-court-cycle redemarrage; FAULT: Etat de defaut *)

{attribute 'qualified_only'}
{attribute 'strict'}
TYPE E_WinchFinalInterlockState : (DISABLED := 0, READY := 1, WAIT_BRAKE_COMMAND_CONFIRMATION := 2, WAIT_STEP_DELAY := 3, WAIT_RESTART_DELAY := 4, FAULT := 5);
END_TYPE

{attribute 'qualified_only'}
VAR_GLOBAL  (* GVL_Troubleshooting - ═══════════════════════════════════════════════════════════════ 🕵️‍♂️ GVL_Troubleshooting — GVL Globale de Recherche de Pannes (Orientée Fonctions & Contexte) ─────────────────────────────────────────────────────────────── ⚙️ Emplacement : CODE/K_DEPANNAGE/GVL_Troubleshooting.st 🎨 Structurée par CONTEXTE GLOBAL MACHINE + FONCTIONS MÉTIER (Utilisation Opérateur). 💬 Permet de localiser en 3 secondes l'environnement et le blocage d'une action. ═══════════════════════════════════════════════════════════════ *)
  ContexteMachineGlobal : ST_ChainContextGlobal;  (* 🌐 0. Contexte Global Machine (Mode, Simu, Commande, Bypass) *)
  LevageSynchroniseM1M2 : ST_ChainWinchSync;  (* 🛗 1. Levage Synchronisé M1+M2 (Mode Couplé Nominal) *)
  LevageUnitaireM1 : ST_ChainWinch;  (* 🛗 2. Levage Unitaire M1 (Treuil Retenue) *)
  LevageUnitaireM2 : ST_ChainWinch;  (* 🛗 3. Levage Unitaire M2 (Treuil Benne) *)
  BenneOuvertureFermeture : ST_ChainBucket;  (* 🪣 4. Ouverture / Fermeture Benne *)
  TranslationPontM3 : ST_ChainTranslation;  (* ↔️ 5. Translation Pont M3 (Variateur AC600) *)
  AssistanceDragage : ST_ChainDredgingAssist;  (* 🌊 5bis. Assistance Plongée/Extraction/Vidage Trémie *)
  CycleSemiAuto : ST_ChainCycleSemiAuto;  (* 🔄 6. Séquenceur de Cycle Semi-Automatique (X0 à X13) *)
  HomingM1 : ST_HomingChecklist;  (* 🎯 Diagnostic chronologique Homing M1 (Treuil Retenue) *)
  HomingM2 : ST_HomingChecklist;  (* 🎯 Diagnostic chronologique Homing M2 (Treuil Benne) *)
  Safety : ST_SafetyChecklist;  (* 🛡️ Diagnostic chronologique Chaîne de Sécurité & Réarmement AU *)
  Joystick : ST_JoystickChecklist;  (* 🕹️ Diagnostic chronologique Bus CANopen & Homme-Mort Joystick *)
  MotionM1 : ST_MotionChecklist;  (* ⚙️ Diagnostic chronologique Mouvement M1 (Treuil Retenue) *)
  MotionM2 : ST_MotionChecklist;  (* ⚙️ Diagnostic chronologique Mouvement M2 (Treuil Benne) *)
  MotionM3 : ST_MotionChecklist;  (* ⚙️ Diagnostic chronologique Mouvement M3 (Translation) *)
  Inputs : ST_HardwareImage;  (* 📥 Image complète des entrées réelles / qualifiées / simulées *)
END_VAR
